// LS Electric XG5000 project: Project
// PLC LSPLC

PROGRAM NewProgram (task: 스캔 프로그램)

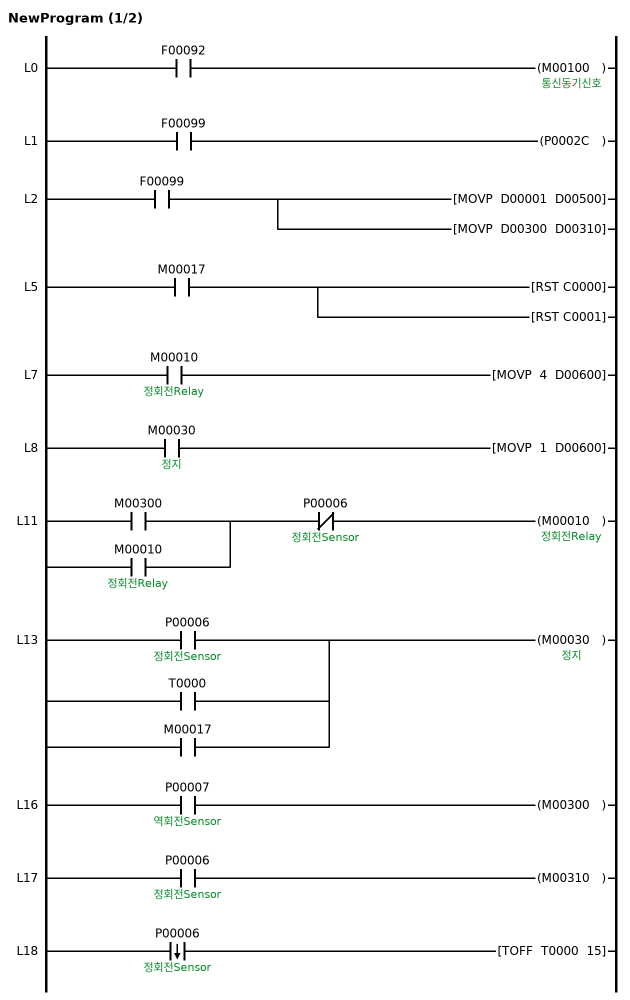
; L0
LOAD      F00092
OUT       M00100	// 통신동기신호
; L1
LOAD      F00099
OUT       P0002C
; L2
LOAD      F00099
MOVP      D00001 D00500
MOVP      D00300 D00310
; L5
LOAD      M00017
RST       C0000
RST       C0001
; L7
LOAD      M00010	// 정회전Relay
MOVP      4 D00600
; L8
LOAD      M00030	// 정지
MOVP      1 D00600
; L11
LOAD      M00300
OR        M00010	// 정회전Relay
AND NOT   P00006	// 정회전Sensor
OUT       M00010	// 정회전Relay
; L13
LOAD      P00006	// 정회전Sensor
OR        T0000
OR        M00017
OUT       M00030	// 정지
; L16
LOAD      P00007	// 역회전Sensor
OUT       M00300
; L17
LOAD      P00006	// 정회전Sensor
OUT       M00310
; L18
LOADN     P00006	// 정회전Sensor
TOFF      T0000 15

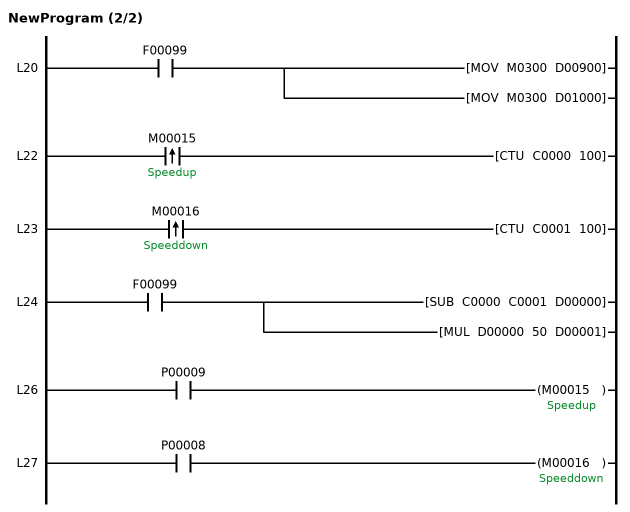
; L20
LOAD      F00099
MOV       M0300 D00900
MOV       M0300 D01000
; L22
LOADP     M00015	// Speedup
CTU       C0000 100
; L23
LOADP     M00016	// Speeddown
CTU       C0001 100
; L24
LOAD      F00099
SUB       C0000 C0001 D00000
MUL       D00000 50 D00001
; L26
LOAD      P00009
OUT       M00015	// Speedup
; L27
LOAD      P00008
OUT       M00016	// Speeddown

VARIABLES AND COMMENTS (devices not used above)
M00000	BIT	MotorStart
P0000A	BIT	stopsw
M00020	BIT	역회전Relay